// Mitsubishi GX Works2 project: Final   PLC: FX1S
// SA

PROGRAM MAIN
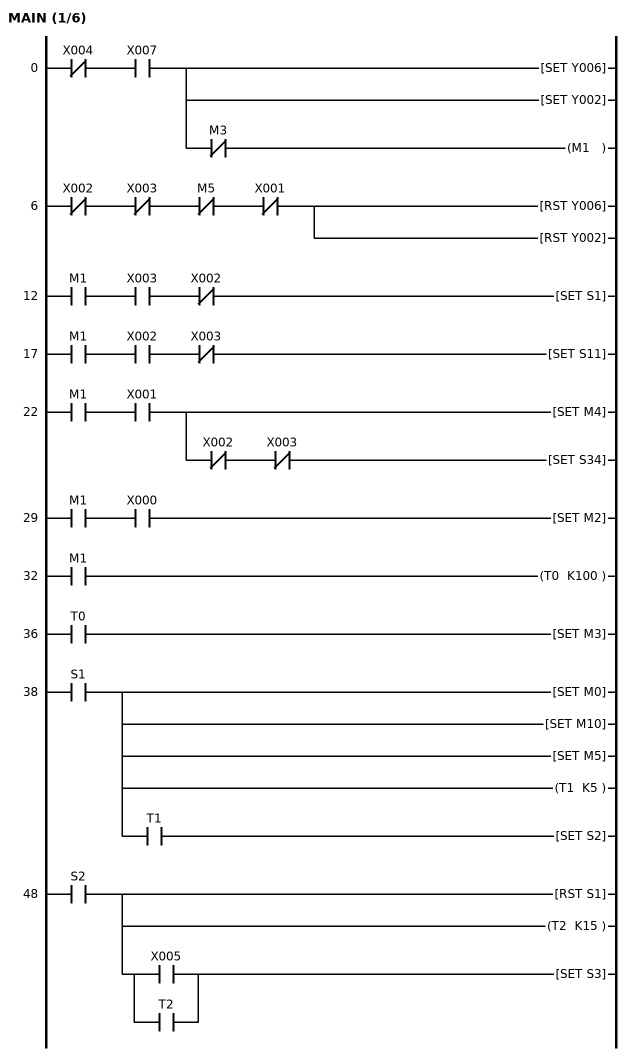
0     LDI     X004
      AND     X007
      SET     Y006
      SET     Y002
      ANI     M3
      OUT     M1
6     LDI     X002
      ANI     X003
      ANI     M5
      ANI     X001
      RST     Y006
      RST     Y002
12    LD      M1
      AND     X003
      ANI     X002
      SET     S1
17    LD      M1
      AND     X002
      ANI     X003
      SET     S11
22    LD      M1
      AND     X001
      SET     M4
      ANI     X002
      ANI     X003
      SET     S34
29    LD      M1
      AND     X000
      SET     M2
32    LD      M1
      OUT     T0 K100
36    LD      T0
      SET     M3
38    LD      S1
      SET     M0
      SET     M10
      SET     M5
      OUT     T1 K5
      AND     T1
      SET     S2
48    LD      S2
      RST     S1
      OUT     T2 K15
      LD      X005
      OR      T2
      ANB
      SET     S3
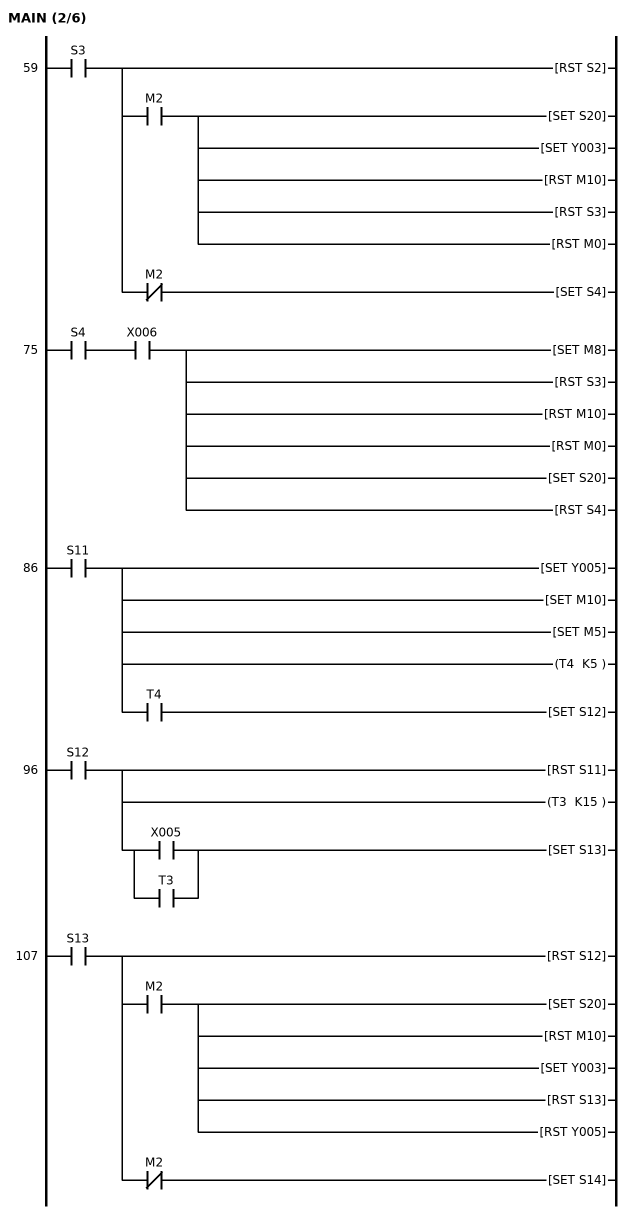
59    LD      S3
      RST     S2
      MPS
      AND     M2
      SET     S20
      SET     Y003
      RST     M10
      RST     S3
      RST     M0
      MPP
      ANI     M2
      SET     S4
75    LD      S4
      AND     X006
      SET     M8
      RST     S3
      RST     M10
      RST     M0
      SET     S20
      RST     S4
86    LD      S11
      SET     Y005
      SET     M10
      SET     M5
      OUT     T4 K5
      AND     T4
      SET     S12
96    LD      S12
      RST     S11
      OUT     T3 K15
      LD      X005
      OR      T3
      ANB
      SET     S13
107   LD      S13
      RST     S12
      MPS
      AND     M2
      SET     S20
      RST     M10
      SET     Y003
      RST     S13
      RST     Y005
      MPP
      ANI     M2
      SET     S14
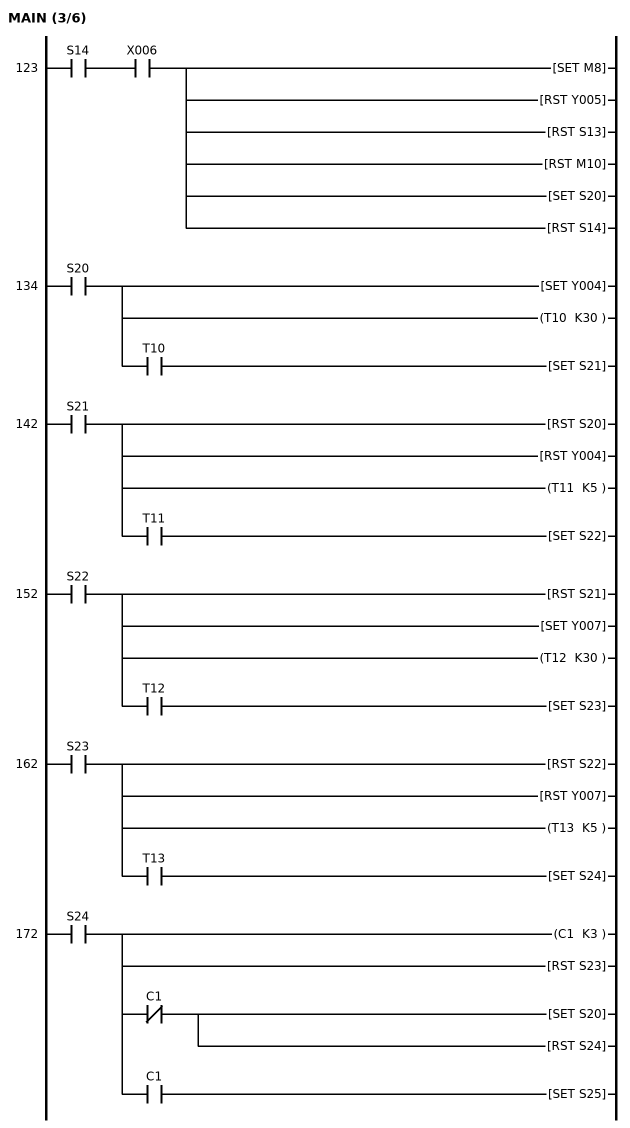
123   LD      S14
      AND     X006
      SET     M8
      RST     Y005
      RST     S13
      RST     M10
      SET     S20
      RST     S14
134   LD      S20
      SET     Y004
      OUT     T10 K30
      AND     T10
      SET     S21
142   LD      S21
      RST     S20
      RST     Y004
      OUT     T11 K5
      AND     T11
      SET     S22
152   LD      S22
      RST     S21
      SET     Y007
      OUT     T12 K30
      AND     T12
      SET     S23
162   LD      S23
      RST     S22
      RST     Y007
      OUT     T13 K5
      AND     T13
      SET     S24
172   LD      S24
      OUT     C1 K3
      RST     S23
      MPS
      ANI     C1
      SET     S20
      RST     S24
      MPP
      AND     C1
      SET     S25
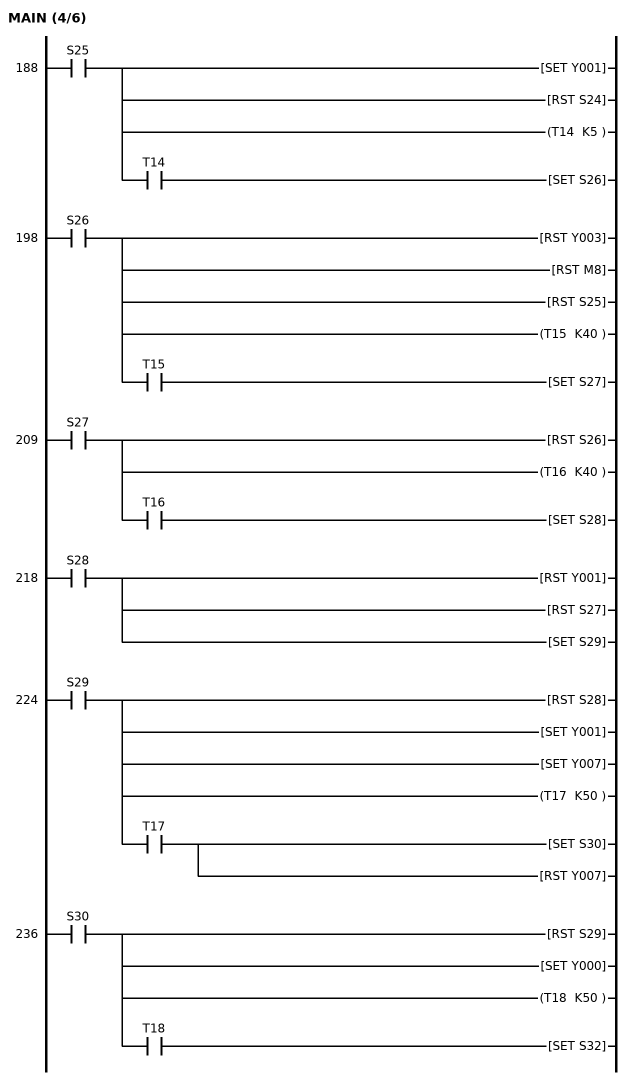
188   LD      S25
      SET     Y001
      RST     S24
      OUT     T14 K5
      AND     T14
      SET     S26
198   LD      S26
      RST     Y003
      RST     M8
      RST     S25
      OUT     T15 K40
      AND     T15
      SET     S27
209   LD      S27
      RST     S26
      OUT     T16 K40
      AND     T16
      SET     S28
218   LD      S28
      RST     Y001
      RST     S27
      SET     S29
224   LD      S29
      RST     S28
      SET     Y001
      SET     Y007
      OUT     T17 K50
      AND     T17
      SET     S30
      RST     Y007
236   LD      S30
      RST     S29
      SET     Y000
      OUT     T18 K50
      AND     T18
      SET     S32
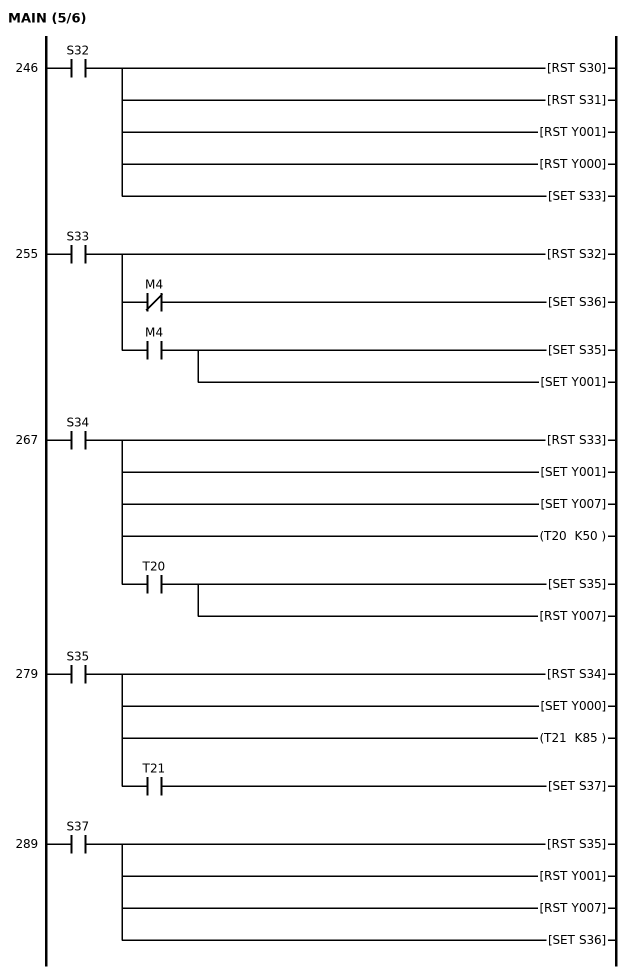
246   LD      S32
      RST     S30
      RST     S31
      RST     Y001
      RST     Y000
      SET     S33
255   LD      S33
      RST     S32
      MPS
      ANI     M4
      SET     S36
      MPP
      AND     M4
      SET     S35
      SET     Y001
267   LD      S34
      RST     S33
      SET     Y001
      SET     Y007
      OUT     T20 K50
      AND     T20
      SET     S35
      RST     Y007
279   LD      S35
      RST     S34
      SET     Y000
      OUT     T21 K85
      AND     T21
      SET     S37
289   LD      S37
      RST     S35
      RST     Y001
      RST     Y007
      SET     S36
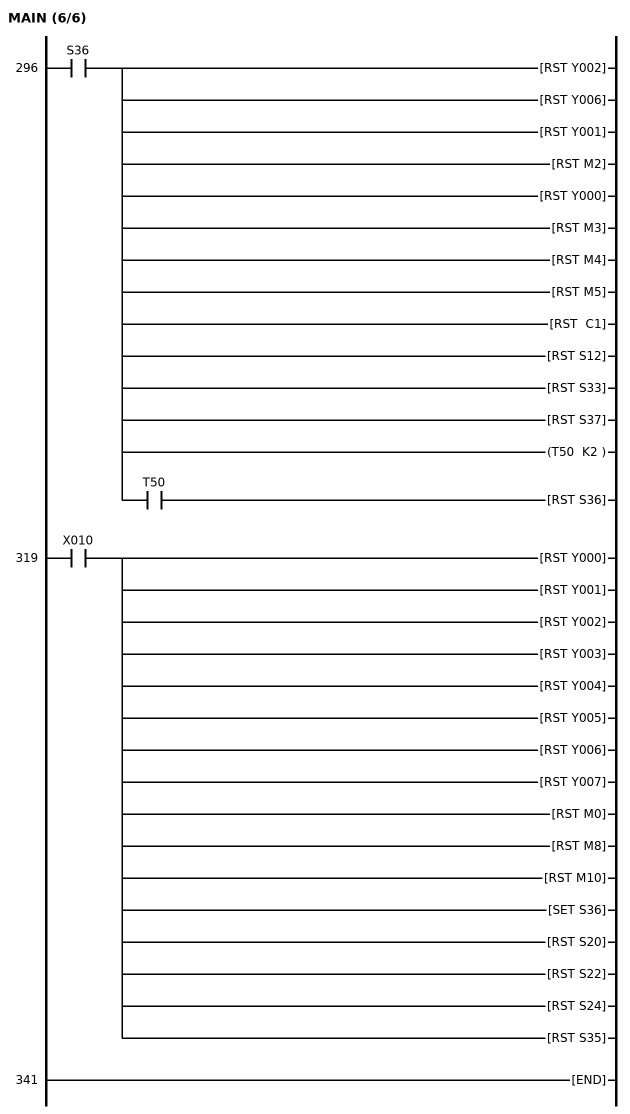
296   LD      S36
      RST     Y002
      RST     Y006
      RST     Y001
      RST     M2
      RST     Y000
      RST     M3
      RST     M4
      RST     M5
      RST     C1
      RST     S12
      RST     S33
      RST     S37
      OUT     T50 K2
      AND     T50
      RST     S36
319   LD      X010
      RST     Y000
      RST     Y001
      RST     Y002
      RST     Y003
      RST     Y004
      RST     Y005
      RST     Y006
      RST     Y007
      RST     M0
      RST     M8
      RST     M10
      SET     S36
      RST     S20
      RST     S22
      RST     S24
      RST     S35
341   END
END_PROGRAM
